Staubli VAL3: JTP.pgx

program JTP()
  local num l_ni
begin
  //建立坐标系
  setFrame(pt1,pt2,pt3,frmaster)
  //数据转换

  for l_ni=0 to nSize-1
    pdemo[l_ni]=jointToPoint(t2,frmaster,A130:ptRoutingPath[l_ni])
  endFor
end
